TEXTLIST TL_E_CTRL_MOVER
  0 = 'MOVER_NULL'
  1 = 'MOVER_ENABLE'
  2 = 'MOVER_DISABLE'
  4 = 'MOVER_MOVE_TO_POS_CA'
  5 = 'MOVER_SEND_TO_POS_CA'
  6 = 'MOVER_HALT'
  7 = 'MOVER_GEAR_IN'
  8 = 'MOVER_GEAR_IN_POS_CA'
  9 = 'MOVER_GEAR_OUT'
  10 = 'MOVER_RESET'
  3 = 'MOVER_MOVE_TO_POS'
   = ''
END_TEXTLIST

(* stored: Version 1.1.0.1, ProductVersion 3.1.4026.18
   TextList TL_E_CTRL_MOVER: Id {ade39097-efc5-4b6c-820d-e3559708dee9} *)
